// TIA Portal V16 export
// export: Created 2024-05-10T06:46:45.9034077Z, ExportSetting WithDefaults, DisplayName Totally Integrated Automation Portal, DisplayVersion V16, DisplayName TIA Portal Version Control Interface, DisplayVersion V16, DisplayName TIA Portal Openness, DisplayVersion V16, DisplayName STEP 7 Professional, DisplayVersion V16, DisplayName STEP 7 Safety, DisplayVersion V16, DisplayName WinCC Professional, DisplayVersion V16
VAR_GLOBAL   // PLC tag table "101生产数据变量表"
   当前日期年 AT %MW700 : Int;
   当前日期月 AT %MW702 : Int;
   当前日期日 AT %MW704 : Int;
   当前日期时 AT %MW706 : Int;
   当前日期分 AT %MW708 : Int;
   当前日期秒 AT %MW710 : Int;
   开机日期年 AT %MW720 : Int;
   开机日期月 AT %MW722 : Int;
   开机日期日 AT %MW724 : Int;
   开机日期时 AT %MW726 : Int;
   开机日期分 AT %MW728 : Int;
   开机日期秒 AT %MW730 : Int;
   "运行时间(H)" AT %MW740 : Int;
   "运行时间(M)" AT %MW742 : Int;
   "停止时间(H)" AT %MW744 : Int;
   "停止时间(M)" AT %MW746 : Int;
   "故障时间(H)" AT %MW748 : Int;
   "故障时间(M)" AT %MW750 : Int;
   生产数量 AT %MD760 : DInt;
   OK数量 AT %MD764 : DInt;
   NG数量 AT %MD768 : DInt;
   累计数量 AT %MD772 : DInt;
   实时节拍 AT %MW780 : Int;
   工作节拍 AT %MW782 : Int;
   "开机时间(H)" AT %MW732 : Int;
   "开机时间(M)" AT %MW734 : Int;
   "稼动率%" AT %MW752 : Int;
   "合格率%" AT %MW776 : Int;
   PPM AT %MW778 : Int;
   设置日期年 AT %MW800 : Int;
   设置日期月 AT %MW802 : Int;
   设置日期日 AT %MW804 : Int;
   设置日期时 AT %MW806 : Int;
   设置日期分 AT %MW808 : Int;
   设置日期秒 AT %MW810 : Int;
   日期设置通知 AT %M812.0 : Bool;
END_VAR
